FUNCTION PunktErsetztKomma : STRING
VAR_INPUT
	in : STRING;
END_VAR
VAR
END_VAR

PunktErsetztKomma:= REPLACE (in,'.',1,FIND (in,','));

END_FUNCTION

(* stored: Version 1.1.0.1, ProductVersion 3.1.4019.2
   POU PunktErsetztKomma: Id {e8da6946-1916-4bb7-b53a-677c6dcf85d9}, SpecialFunc None *)
